FUNCTION_BLOCK PUBLIC FB_ErrorLogger
VAR_INPUT
	
END_VAR
VAR_OUTPUT
	
END_VAR
VAR
	
END_VAR

END_FUNCTION_BLOCK

(* stored: Version 1.1.0.1, ProductVersion 3.1.4024.14
   POU FB_ErrorLogger: Id {f83db9ac-a4cd-4080-900e-a00207e1af95}, SpecialFunc None *)
